// LS Electric XG5000 project: timer
// PLC NewPLC
// module base 0 slot 0: 입출력 모듈:XBC-DR20S (DC 24V 입력 12점, 릴레이 출력 8점)

PROGRAM NewProgram (task: 스캔 프로그램)

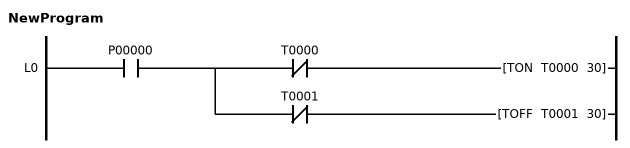
; L0
LOAD      P00000
MPUSH
AND NOT   T0000
TON       T0000 30
MPOP
AND NOT   T0001
TOFF      T0001 30